// TIA Portal project "ERA_TemplateDemo" (V15.1)

(* hardware
DEVICE "S71500/ET200MP-Station_1"  S7-1500 station
   slot 0: "Profilschiene_0"  Rack  6ES7 590-1***0-0AA0
   slot 0: "PM 190W 120/230VAC"  PM 190W 120/230VAC  6EP1333-4BA00
   slot 1: "PLC_1"  CPU 1512C-1 PN  6ES7 512-1CK01-0AB0  V2.6
      slot 3: "CPU-Display_1"  6ES7591-1AA00-0AA0
   slot 2: "AQ 4xU/I ST_1"  AQ 4xU/I ST  6ES7 532-5HD00-0AB0  V2.2
*)

// ===== PLC "PLC_1"  CPU 1512C-1 PN =====

VAR_GLOBAL   // PLC tag table "Standard-Variablentabelle"
   "L1" AT %IW0 : Int;   // Füllstand
   "F1" AT %IW2 : Int;   // Durchfluss, regelbare Pumpe
   "P1" AT %IW4 : Int;   // Druck, regelbare Pumpe
   "T1" AT %IW6 : Int;   // Temperatur
   "FC1" AT %QW0 : Int;   // Stellsignal FU für Pumpe M3
   "FC2" AT %QW2 : Int;   // Stellsignal regelbares Ventil
   "B1" AT %I12.0 : Bool;   // Oberer Füllstandsschalter
   "B2" AT %I12.1 : Bool;   // Mittlerer Füllstandsschalter
   "B3" AT %I12.2 : Bool;   // Unterer Füllstandsschalter
   "HS1" AT %I12.3 : Bool;   // Schalter HS1
   "HS2" AT %I12.4 : Bool;   // Schalter HS2
   "HS3" AT %I12.5 : Bool;   // Schalter HS3
   "HS4" AT %I12.6 : Bool;   // Taster HS4
   "HS5" AT %I12.7 : Bool;   // Taster HS5
   "M1" AT %Q6.0 : Bool;   // Pumpe 1, Zulaufpumpe
   "M2" AT %Q6.1 : Bool;   // Pumpe 2, Zulaufpumpe
   "M3" AT %Q6.2 : Bool;   // Pumpe 3, Ablauf
   "M4" AT %Q6.3 : Bool;   // Pumpe 4, Umwälzpumpe
   "LED1" AT %Q6.4 : Bool;   // Lampe 1, Rot
   "LED2" AT %Q6.5 : Bool;   // Lampe 2, Gelb
   "LED3" AT %Q6.6 : Bool;   // Lampe 3, Grün
   "Y1" AT %Q6.7 : Bool;   // Ventil 4
   "Cao" AT %Q7.0 : Bool;
   "Tou" AT %Q7.1 : Bool;
END_VAR

DATA_BLOCK "Programm_DB"   // DB1
{ S7_Optimized_Access := 'TRUE' }
VERSION : 0.1
// stored: InstanceOfName Programm
"Programm"
BEGIN
END_DATA_BLOCK

FUNCTION_BLOCK "Programm"   // FB1, LAD
{ S7_Optimized_Access := 'TRUE' }
VERSION : 0.1
   VAR_TEMP
      Pendeln : Bool;
      Zulauf : Bool;
      ablauf : Bool;
   END_VAR
BEGIN

REGION Network 1: BEISPIEL
   // Dieses Netzwerk dient nur zur Veranschaulichung. Bitte loeschen bzw. ueberschreiben.
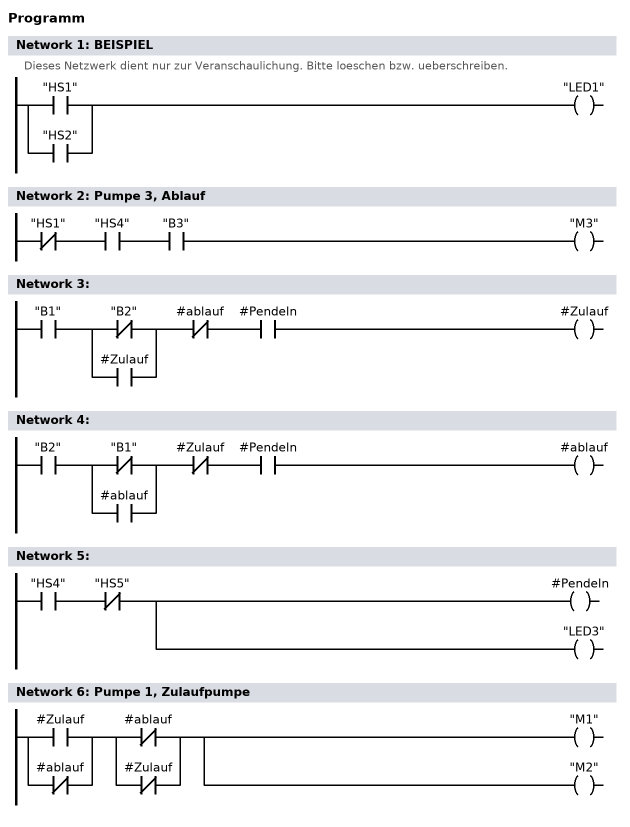
   RUNG wire#powerrail
      Contact( "HS1" )
      wire#w1
      Coil( "LED1" )
   END_RUNG
   RUNG wire#powerrail
      Contact( "HS2" )
   END_RUNG wire#w1
   // the same network as SCL:
   "LED1" := "HS1" OR "HS2";
END_REGION

REGION Network 2: Pumpe 3, Ablauf
   RUNG wire#powerrail
      I_Contact( "HS1" )
      Contact( "HS4" )
      Contact( "B3" )
      Coil( "M3" )
   END_RUNG
   // the same network as SCL:
   "M3" := NOT "HS1" AND "HS4" AND "B3";
END_REGION

REGION Network 3
   RUNG wire#powerrail
      Contact( "B1" )
      wire#w1
      I_Contact( "B2" )
      wire#w2
      I_Contact( #ablauf )
      Contact( #Pendeln )
      Coil( #Zulauf )
   END_RUNG
   RUNG wire#w1
      Contact( #Zulauf )
   END_RUNG wire#w2
   // the same network as SCL:
   #Zulauf := "B1" AND (NOT "B2" OR #Zulauf) AND NOT #ablauf AND #Pendeln;
END_REGION

REGION Network 4
   RUNG wire#powerrail
      Contact( "B2" )
      wire#w1
      I_Contact( "B1" )
      wire#w2
      I_Contact( #Zulauf )
      Contact( #Pendeln )
      Coil( #ablauf )
   END_RUNG
   RUNG wire#w1
      Contact( #ablauf )
   END_RUNG wire#w2
   // the same network as SCL:
   #ablauf := "B2" AND (NOT "B1" OR #ablauf) AND NOT #Zulauf AND #Pendeln;
END_REGION

REGION Network 5
   RUNG wire#powerrail
      Contact( "HS4" )
      I_Contact( "HS5" )
      wire#w1
      Coil( #Pendeln )
   END_RUNG
   RUNG wire#w1
      Coil( "LED3" )
   END_RUNG
   // the same network as SCL:
   #Pendeln := "HS4" AND NOT "HS5";
   "LED3" := #Pendeln;
END_REGION

REGION Network 6: Pumpe 1, Zulaufpumpe
   RUNG wire#powerrail
      Contact( #Zulauf )
      wire#w1
      I_Contact( #ablauf )
      wire#w2
      Coil( "M1" )
   END_RUNG
   RUNG wire#powerrail
      I_Contact( #ablauf )
   END_RUNG wire#w1
   RUNG wire#w1
      I_Contact( #Zulauf )
   END_RUNG wire#w2
   RUNG wire#w2
      Coil( "M2" )
   END_RUNG
   // the same network as SCL:
   "M1" := (#Zulauf OR NOT #ablauf) AND (NOT #ablauf OR NOT #Zulauf);
   "M2" := "M1";
END_REGION
END_FUNCTION_BLOCK

ORGANIZATION_BLOCK "Main"   // OB1, LAD, ProgramCycle
TITLE = "Main Program Sweep (Cycle)"
{ S7_Optimized_Access := 'TRUE' }
VERSION : 0.1
   VAR_INPUT
      Initial_Call : Bool;   // Initial call of this OB
      Remanence : Bool;   // =True, if remanent data are available
   END_VAR
BEGIN

REGION Network 1
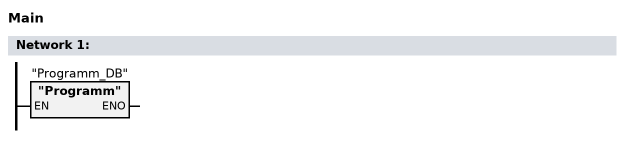
   RUNG wire#powerrail
      "Programm_DB"()
   END_RUNG
   // the same network as SCL:
   "Programm_DB"();   // "Programm"
END_REGION
END_ORGANIZATION_BLOCK